FUNCTION_BLOCK Fb_BindControlVars
VAR_INPUT
	AdvancedControl : BOOL;
END_VAR

VAR_IN_OUT
	SystemControlVars : ST_System_Control;
	ExtControlVars		: ST_ExtController_get;
END_VAR

VAR
	defaults			: ST_Softsettings;
	ftrig_AdvancedControl : F_trig;
	rTrig_AdvancedControl : R_Trig;
	
	b_defaultsRestored	: BOOL;
END_VAR

VAR
	WoE_Start		:	WriteOnEdge;
	WoE_Stop		:	WriteOnEdge;
	WoE_Activate	:	WriteOnEdge;
	WoE_Shutdown	:	WriteOnEdge;
	WoE_ClearHistory	:	WriteOnEdge;
	WoE_EMstop		:	WriteOnEdge;
	WoE_DehumStart	:	WriteOnEdge;
	WoE_Reset		:	WriteOnEdge;
END_VAR
VAR // added by the converter: edge detectors and wires of the graphical bodies
    _rt1, _rt2, _rt3, _rt4, _rt5, _rt6, _rt7, _rt8 : R_TRIG;
END_VAR

ftrig_AdvancedControl(CLK:= advancedcontrol);
IF ftrig_advancedControl.Q THEN
	RestoreDefaults(defaults, Systemcontrolvars.SoftSettings);
END_IF

//advanced control, all IO coupled
IF advancedcontrol THEN
	SystemControlVars.SoftSettings := ExtControlVars.SoftSettings;
	SystemControlVars.Operation := ExtControlVars.Operation;
ELSE
	Storedefaults(defaults, Systemcontrolvars.SoftSettings);
	//Basic control, only specific IO coupled
	Systemcontrolvars.softsettings.system.b_EcoModeEnable := ExtControlVars.SoftSettings.system.b_EcoModeEnable;
	SystemControlvars.operation.system.b_PFsetEnable := ExtControlVars.Operation.system.b_PFsetEnable;
	SystemControlvars.operation.system.r_PFset := ExtControlVars.Operation.system.r_PFset;
	SystemControlvars.operation.system.r_Pset:= ExtControlVars.Operation.system.r_Pset;
	SystemControlvars.operation.system.r_Qset:= ExtControlVars.Operation.system.r_Qset;
	SystemControlvars.softsettings.PSB.setpointTimeslot1 := ExtControlVars.softsettings.PSB.setpointTimeslot1;
END_IF

a_ControlCommands();

ACTION a_ControlCommands:
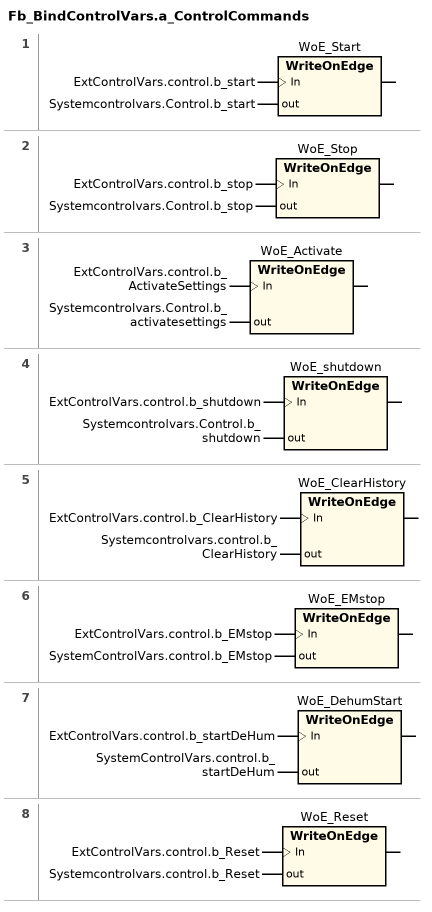
// NETWORK 1
_rt1(CLK := ExtControlVars.control.b_start);
WoE_Start(In := _rt1.Q, out := Systemcontrolvars.Control.b_start); // WriteOnEdge

// NETWORK 2
_rt2(CLK := ExtControlVars.control.b_stop);
WoE_Stop(In := _rt2.Q, out := Systemcontrolvars.Control.b_stop); // WriteOnEdge

// NETWORK 3
_rt3(CLK := ExtControlVars.control.b_ActivateSettings);
WoE_Activate(In := _rt3.Q, out := Systemcontrolvars.Control.b_activatesettings); // WriteOnEdge

// NETWORK 4
_rt4(CLK := ExtControlVars.control.b_shutdown);
WoE_shutdown(In := _rt4.Q, out := Systemcontrolvars.Control.b_shutdown); // WriteOnEdge

// NETWORK 5
_rt5(CLK := ExtControlVars.control.b_ClearHistory);
WoE_ClearHistory(In := _rt5.Q, out := Systemcontrolvars.control.b_ClearHistory); // WriteOnEdge

// NETWORK 6
_rt6(CLK := ExtControlVars.control.b_EMstop);
WoE_EMstop(In := _rt6.Q, out := SystemControlVars.control.b_EMstop); // WriteOnEdge

// NETWORK 7
_rt7(CLK := ExtControlVars.control.b_startDeHum);
WoE_DehumStart(In := _rt7.Q, out := SystemControlVars.control.b_startDeHum); // WriteOnEdge

// NETWORK 8
_rt8(CLK := ExtControlVars.control.b_Reset);
WoE_Reset(In := _rt8.Q, out := Systemcontrolvars.control.b_Reset); // WriteOnEdge
END_ACTION

METHOD RestoreDefaults
VAR_IN_OUT
	defaults 		: ST_Softsettings;
	softsettings	: ST_Softsettings;
END_VAR
IF memcmp(pBuf1 := ADR(defaults), pBuf2:= ADR(softsettings), n:= SIZEOF(defaults)) <> 0 THEN
	softsettings := defaults;
END_IF
END_METHOD

METHOD StoreDefaults : BOOL
VAR_IN_OUT
	defaults 		: ST_Softsettings;
	softsettings	: ST_Softsettings;
END_VAR
StoreDefaults := FALSE;

IF memcmp(pBuf1 := ADR(defaults), pBuf2:= ADR(softsettings), n:= SIZEOF(defaults)) <> 0 THEN
	defaults := softsettings;
ELSE
	StoreDefaults := TRUE;
END_IF
END_METHOD

END_FUNCTION_BLOCK

(* stored: Version 1.1.0.1, ProductVersion 3.1.4026.18
   POU Fb_BindControlVars: Id {2582c493-ebec-4155-9106-ed507abe1cad}, SpecialFunc None
   Action a_ControlCommands: Id {0d40d958-265e-4b54-b1c8-8e23b865c215}
   Method RestoreDefaults: Id {bd8642b8-6375-4475-935d-96b5f2275b03}
   Method StoreDefaults: Id {dcd571db-791f-447d-ae89-e1b6e012a7b0} *)
